Universal Robots URScript: Programa_iniciales.script

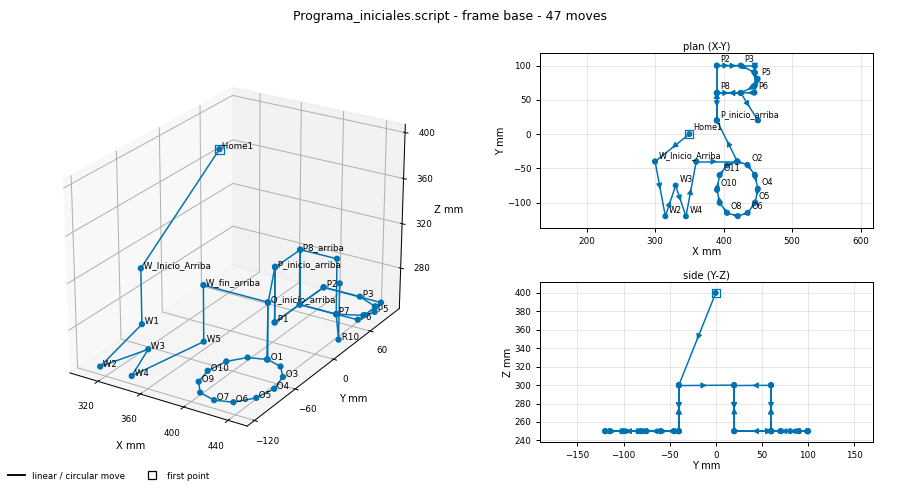
[picture p0: tool path of Programa_iniciales.script in frame base, 47 of 47 moves have a stored position in this frame; points joined in program order, loops and branches not executed]
def Programa_iniciales():
  set_standard_analog_input_domain(0, 1)
  set_standard_analog_input_domain(1, 1)
  set_tool_analog_input_domain(0, 1)
  set_tool_analog_input_domain(1, 1)
  set_analog_outputdomain(0, 0)
  set_analog_outputdomain(1, 0)
  set_input_actions_to_default()
  step_count_ec848798_e229_4b4f_a1ae_adc986fa359f = 0.0
  thread Step_Counter_Thread_7c991857_774f_46ef_b6ad_21fa12a4a815():
    while (True):
      step_count_ec848798_e229_4b4f_a1ae_adc986fa359f = step_count_ec848798_e229_4b4f_a1ae_adc986fa359f + 1.0
      sync()
    end
  end
  run Step_Counter_Thread_7c991857_774f_46ef_b6ad_21fa12a4a815()
  set_safety_mode_transition_hardness(1)
  set_gravity([0.0, 0.0, 9.82])
  set_tcp(p[0.0,0.0,0.0,0.0,0.0,0.0])
  set_payload(0.5, [0.0, 0.0, 0.05])
  set_tool_voltage(0)
  # begin: URCap Installation Node
  #   Source: External Control, 1.0.5, FZI Research Center for Information Technology
  #   Type: External Control
  # end: URCap Installation Node
  $ 1 "Robot Program"
  $ 2 "MoveJ"
  $ 3 "Home1" "breakAfter"
  movej(get_inverse_kin(p[.349999980891, -.000000009801, .400000017349, -.000000033462, 3.141185121458, .000000117007], qnear=[0.3171784579753876, -1.1990464369403284, -1.949850861226217, -1.5631044546710413, 1.5706692934036255, 1.887974739074707]), a=1.3962634015954636, v=1.0471975511965976)
  $ 4 "Popup: Se simulara la letra W del integrante con iniciales WO"
  popup("Se simulara la letra W del integrante con iniciales WO", "Message", False, False, blocking=True)
  $ 5 "MoveL"
  $ 6 "W_Inicio_Arriba" "breakAfter"
  movel(p[.300000006338, -.039999994203, .299999982186, -.000000042425, 3.141185498596, -.000000117222], a=0.1, v=0.05)
  $ 7 "W1" "breakAfter"
  movel(p[.299999982052, -.039999999482, .250000163231, .000000089212, -3.141185111532, .000000044313], a=0.1, v=0.05)
  $ 8 "W2" "breakAfter"
  movel(p[.314978571165, -.119885735890, .250000222850, .000000210688, -3.141185236972, -.000000018331], a=0.1, v=0.05)
  $ 9 "W3" "breakAfter"
  movel(p[.329999781078, -.075000683460, .250000290523, .000000140416, -3.141185369267, -.000000109433], a=0.1, v=0.05)
  $ 10 "W4" "breakAfter"
  movel(p[.344999964915, -.120000038798, .250000382110, .000000023111, -3.141185748465, -.000000023522], a=0.1, v=0.05)
  $ 11 "W5" "breakAfter"
  movel(p[.359987422572, -.040067314232, .250000448595, .000000117557, -3.141185839983, -.000000062155], a=0.1, v=0.05)
  $ 12 "W_fin_arriba" "breakAfter"
  movel(p[.359999959989, -.040000052920, .299961771332, .000000164327, -3.141185816835, -.000000128285], a=0.1, v=0.05)
  $ 13 "Popup: Se simuara la letra O del integrante con las iniciales WO"
  popup("Se simuara la letra O del integrante con las iniciales WO", "Message", False, False, blocking=True)
  $ 14 "O_inicio_arriba" "breakAfter"
  movel(p[.419788570047, -.040000044335, .299999793978, .000000214594, -3.141185534738, -.000000063125], a=0.1, v=0.05)
  $ 15 "O1" "breakAfter"
  movel(p[.419999917058, -.040000053795, .250004926504, .000000120954, -3.141185064517, .000000006105], a=0.1, v=0.05)
  $ 16 "O2" "breakAfter"
  movel(p[.434653232916, -.044884377980, .250004919249, .000000123091, -3.141185211668, -.000000022566], a=0.1, v=0.05)
  $ 17 "O3" "breakAfter"
  movel(p[.445446966144, -.059263265205, .250004952772, .000000186208, -3.141185255982, .000000045285], a=0.1, v=0.05)
  $ 18 "O4" "breakAfter"
  movel(p[.449930417698, -.079682926674, .250004896589, .000000274144, -3.141185060679, -.000000026729], a=0.1, v=0.05)
  $ 19 "O5" "breakAfter"
  movel(p[.446073611035, -.099619437420, .250005016894, .000000338437, -3.141185376305, -.000000038293], a=0.1, v=0.05)
  $ 20 "O6" "breakAfter"
  movel(p[.435084262202, -.114882830431, .250005031565, .000000582440, -3.141185435469, -.000000055791], a=0.1, v=0.05)
  $ 21 "O7" "breakAfter"
  movel(p[.420800825347, -.119728356494, .250005034866, .000000396774, -3.141185342288, .000000009356], a=0.1, v=0.05)
  $ 22 "O8" "breakAfter"
  movel(p[.405118153712, -.115035409827, .249999898594, .000000208175, -3.141184950457, .000000009759], a=0.1, v=0.05)
  $ 23 "O9" "breakAfter"
  movel(p[.394351299380, -.100475032999, .249999898833, .000000206712, -3.141184894393, .000000015377], a=0.1, v=0.05)
  $ 24 "O10" "breakAfter"
  movel(p[.390300586443, -.081414706905, .249999866967, .000000191507, -3.141184905126, .000000094304], a=0.1, v=0.05)
  $ 25 "O11" "breakAfter"
  movel(p[.393996180821, -.060021712830, .249999792795, .000000125993, -3.141184616261, .000000103501], a=0.1, v=0.05)
  $ 26 "O12" "breakAfter"
  movel(p[.404711109579, -.045394352705, .249999739019, .000000051597, -3.141184587955, .000000136852], a=0.1, v=0.05)
  $ 27 "O13" "breakAfter"
  movel(p[.419344114728, -.040231406173, .249999782425, -.000000019456, -3.141184614033, .000000127132], a=0.1, v=0.05)
  $ 28 "O_fin_arriba" "breakAfter"
  movel(p[.419993310231, -.040002366450, .299486772012, .000000050718, -3.141184594291, .000000128539], a=0.1, v=0.05)
  $ 29 "Popup: Se simulara la letra P del integrante con las iniciales PR"
  popup("Se simulara la letra P del integrante con las iniciales PR", "Message", False, False, blocking=True)
  $ 30 "P_inicio_arriba" "breakAfter"
  movel(p[.390033524865, .019932936927, .299999298575, .000000078370, -3.141184381807, .000000258830], a=0.1, v=0.05)
  $ 31 "P1" "breakAfter"
  movel(p[.390000150329, .019999833087, .250141747278, .000000171949, -3.141184342714, .000000208734], a=0.1, v=0.05)
  $ 32 "P2" "breakAfter"
  movel(p[.390000185281, .099856933141, .250000343231, .000000062131, -3.141184382275, .000000156750], a=0.1, v=0.05)
  $ 33 "P3" "breakAfter"
  movel(p[.424920521408, .099999653456, .250000415049, -.000000075398, -3.141184427450, .000000117048], a=0.1, v=0.05)
  $ 34 "P4" "breakAfter"
  movel(p[.444815537589, .090091871580, .250000543034, .000000021498, -3.141184740814, -.000000120629], a=0.1, v=0.05)
  $ 35 "P5" "breakAfter"
  movel(p[.449621531678, .080736743511, .250000386612, -.000000023316, -3.141184525705, .000000052131], a=0.1, v=0.05)
  $ 36 "P6" "breakAfter"
  movel(p[.445095533473, .060428451707, .250000494836, -.000000066545, -3.141184913968, -.000000104001], a=0.1, v=0.05)
  $ 37 "P7" "breakAfter"
  movel(p[.425028053233, .060000596097, .250000416527, -.000000114971, -3.141184678988, -.000000020688], a=0.1, v=0.05)
  $ 38 "P8" "breakAfter"
  movel(p[.390000656123, .060000612308, .250000395659, -.000000164918, -3.141184579954, .000000128479], a=0.1, v=0.05)
  $ 39 "P8_arriba" "breakAfter"
  movel(p[.390000724255, .060000643782, .299774386207, -.000000164918, -3.141184579954, .000000128480], a=0.1, v=0.05)
  $ 40 "Popup: Se simulara la letra R"
  popup("Se simulara la letra R", "Message", False, False, blocking=True)
  $ 41 "R_inicio_arriba" "breakAfter"
  movel(p[.390145372405, .020000020342, .299565054148, -.000000577032, -3.141183480959, .000000796094], a=0.1, v=0.05)
  $ 42 "R1" "breakAfter"
  movel(p[.390145398491, .020000029416, .249999595305, -.000000577032, -3.141183480959, .000000796094], a=0.1, v=0.05)
  $ 43 "R2" "breakAfter"
  movel(p[.390145315227, .099997901777, .249999592019, -.000000593357, -3.141183497419, .000000827397], a=0.1, v=0.05)
  $ 44 "R3" "breakAfter"
  movel(p[.445502614154, .099204640574, .249999638794, -.000000682237, -3.141183599198, .000000775806], a=0.1, v=0.05)
  $ 45 "R4" "breakAfter"
  movel(p[.445502555291, .089942050353, .249999658083, -.000000727511, -3.141183600747, .000000723786], a=0.1, v=0.05)
  $ 46 "R5" "breakAfter"
  movel(p[.445502534435, .071068427127, .249999658465, -.000000583667, -3.141183498535, .000000856205], a=0.1, v=0.05)
  $ 47 "R6" "breakAfter"
  movel(p[.444949646213, .069954087077, .250045519097, -.000000630357, -3.141183291642, .000000820924], a=0.1, v=0.05)
  $ 48 "R7" "breakAfter"
  movel(p[.425100513010, .060050139667, .250045694635, -.000000583162, -3.141183799619, .000000586280], a=0.1, v=0.05)
  $ 49 "R8" "breakAfter"
  movel(p[.390453554567, .060050128720, .250045719978, -.000000633084, -3.141183764059, .000000681539], a=0.1, v=0.05)
  $ 50 "R8_arriba" "breakAfter"
  movel(p[.390000454526, .060000033614, .299944119617, -.000000492697, -3.141183714247, .000000756128], a=0.1, v=0.05)
  $ 51 "Popup: Se simulara la letra R.Trazo 2:diagonal"
  popup("Se simulara la letra R.Trazo 2:diagonal", "Message", False, False, blocking=True)
  $ 52 "R9_arriba" "breakAfter"
  movel(p[.424753325212, .060000020295, .299999618948, -.000000536354, -3.141183799707, .000000722701], a=0.1, v=0.05)
  $ 53 "R9" "breakAfter"
  movel(p[.424999245618, .060000034730, .250159417871, -.000000489512, -3.141183845743, .000000748072], a=0.1, v=0.05)
  $ 54 "R10" "breakAfter"
  movel(p[.449850685360, .020238857799, .250000898790, -.000000478612, -3.141183811549, .000000698228], a=0.1, v=0.05)
  $ 55 "R_fin_arriba" "breakAfter"
  movel(p[.449999723404, .020000375309, .299918269217, -.000000525345, -3.141183879334, .000000658780], a=0.1, v=0.05)
end
